# EPICS StreamDevice protocol: keithley6221App/src/K6221.proto
Terminator = LF;

getDeviceInfo {
    wait 50;
    ExtraInput = Ignore;
    out "*IDN?";
    in "%40c";
}

getAvailableMemory {
    wait 50;
    ExtraInput = Ignore;
    out "TRAC:FREE?";
    in "%i";
}

QueryConnection {
    wait 50;
    ExtraInput = Ignore;
    out "SOUR:DELta:NVPR?";
    out "%b";
}
